(*
State of a Job.
*)
{attribute 'qualified_only'}
{attribute 'strict'}
TYPE JobState :
(
	Error,
	Idle,
	Enqueue,
	Ready,
	Running,
	Aborted,
	Completed
) BYTE := Idle;
END_TYPE

(* stored: Version 1.1.0.1
   DUT JobState: Id {cb7f1807-8f28-408f-8949-81e30fc2ee8b} *)
